Staubli VAL3: setDefaultType.pgx

public program setDefaultType(num& x_nType[])
begin
  // set the last type used
  saveCycle:nType=x_nType
end
